// SIMATIC S7-200 SMART project (STEP 7-Micro/WIN SMART), CPU CR40

SYMBOL_TABLE 表格 1
启动               M0.4
延时启动             M0.5
延时装置             T37
工件夹持检测虚拟         M0.6
END_SYMBOL_TABLE

SYMBOL_TABLE 系统符号
First_Scan_On    SM0.1    // 仅在第一个扫描周期时接通
Clock_1s         SM0.5    // 针对 1 s 的周期时间，时钟脉冲接通 0.5 s，断开 0.5 s.
END_SYMBOL_TABLE

ORGANIZATION_BLOCK MAIN:OB1
TITLE=主程序
BEGIN
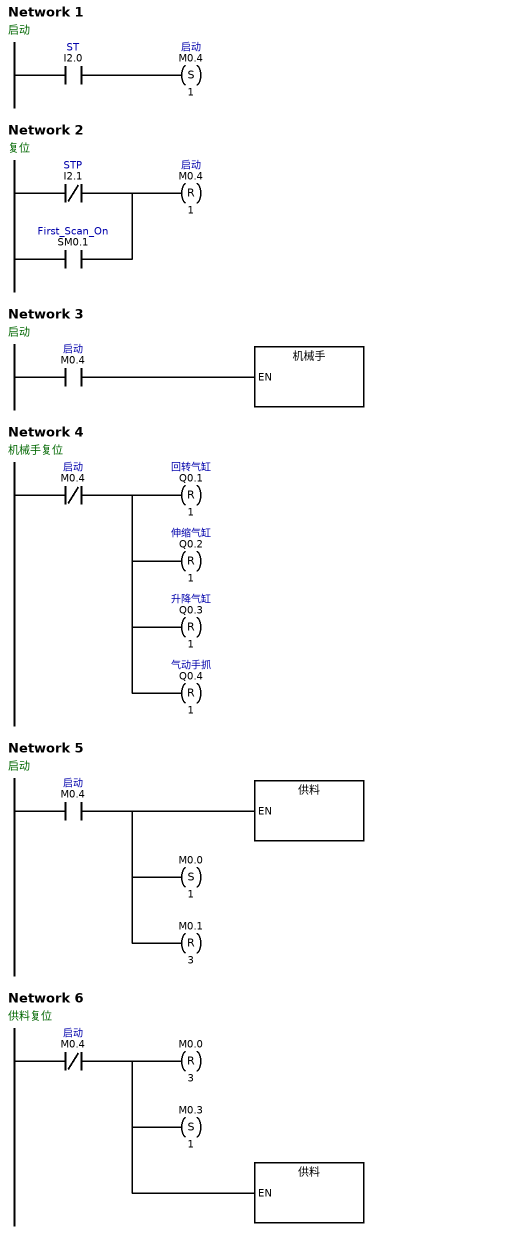
Network 1
// 启动
LD     ST:I2.0
S      启动:M0.4, 1
Network 2
// 复位
LDN    STP:I2.1
O      First_Scan_On:SM0.1
R      启动:M0.4, 1
Network 3
// 启动
LD     启动:M0.4
CALL   机械手:SBR0
Network 4
// 机械手复位
LDN    启动:M0.4
R      回转气缸:Q0.1, 1
R      伸缩气缸:Q0.2, 1
R      升降气缸:Q0.3, 1
R      气动手抓:Q0.4, 1
Network 5
// 启动
LD     启动:M0.4
CALL   供料:SBR3
S      M0.0, 1
R      M0.1, 3
Network 6
// 供料复位
LDN    启动:M0.4
R      M0.0, 3
S      M0.3, 1
CALL   供料:SBR3
END_ORGANIZATION_BLOCK

SUBROUTINE_BLOCK 机械手:SBR0
TITLE=子程序注释
BEGIN
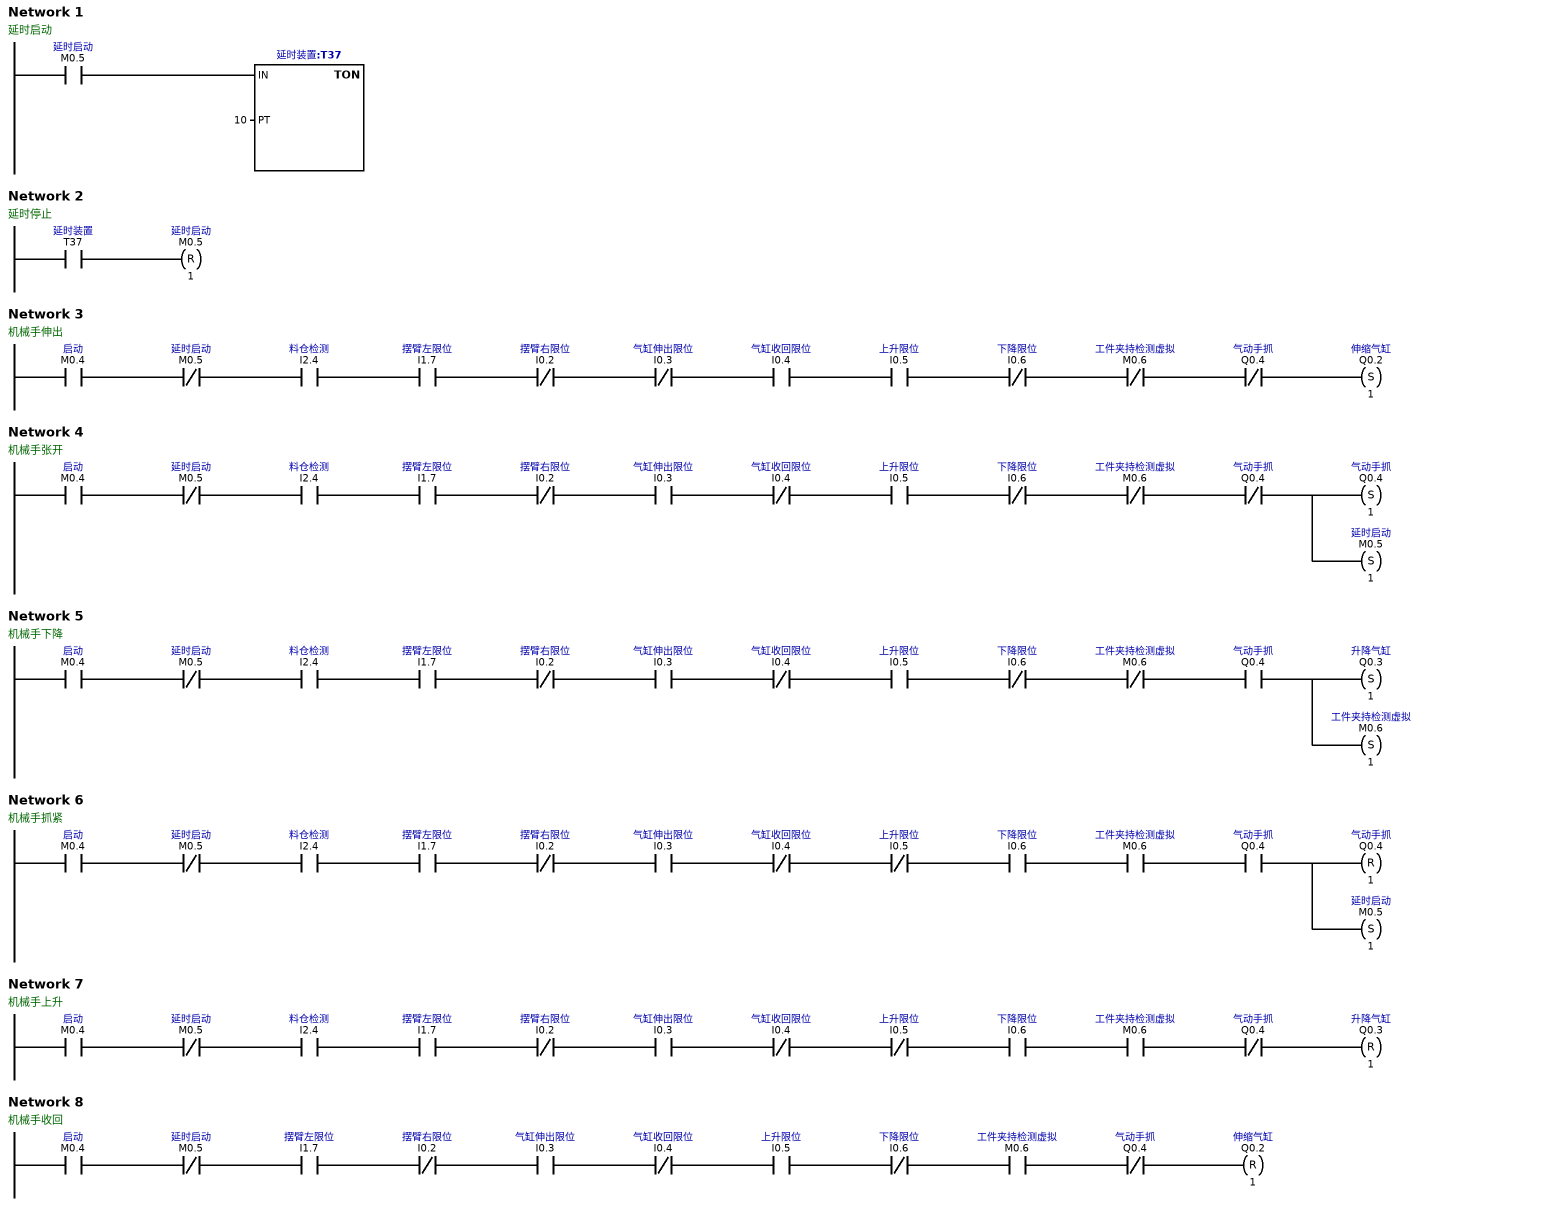
Network 1
// 延时启动
LD     延时启动:M0.5
TON    延时装置:T37, 10
Network 2
// 延时停止
LD     延时装置:T37
R      延时启动:M0.5, 1
Network 3
// 机械手伸出
LD     启动:M0.4
AN     延时启动:M0.5
A      料仓检测:I2.4
A      摆臂左限位:I1.7
AN     摆臂右限位:I0.2
AN     气缸伸出限位:I0.3
A      气缸收回限位:I0.4
A      上升限位:I0.5
AN     下降限位:I0.6
AN     工件夹持检测虚拟:M0.6
AN     气动手抓:Q0.4
S      伸缩气缸:Q0.2, 1
Network 4
// 机械手张开
LD     启动:M0.4
AN     延时启动:M0.5
A      料仓检测:I2.4
A      摆臂左限位:I1.7
AN     摆臂右限位:I0.2
A      气缸伸出限位:I0.3
AN     气缸收回限位:I0.4
A      上升限位:I0.5
AN     下降限位:I0.6
AN     工件夹持检测虚拟:M0.6
AN     气动手抓:Q0.4
S      气动手抓:Q0.4, 1
S      延时启动:M0.5, 1
Network 5
// 机械手下降
LD     启动:M0.4
AN     延时启动:M0.5
A      料仓检测:I2.4
A      摆臂左限位:I1.7
AN     摆臂右限位:I0.2
A      气缸伸出限位:I0.3
AN     气缸收回限位:I0.4
A      上升限位:I0.5
AN     下降限位:I0.6
AN     工件夹持检测虚拟:M0.6
A      气动手抓:Q0.4
S      升降气缸:Q0.3, 1
S      工件夹持检测虚拟:M0.6, 1
Network 6
// 机械手抓紧
LD     启动:M0.4
AN     延时启动:M0.5
A      料仓检测:I2.4
A      摆臂左限位:I1.7
AN     摆臂右限位:I0.2
A      气缸伸出限位:I0.3
AN     气缸收回限位:I0.4
AN     上升限位:I0.5
A      下降限位:I0.6
A      工件夹持检测虚拟:M0.6
A      气动手抓:Q0.4
R      气动手抓:Q0.4, 1
S      延时启动:M0.5, 1
Network 7
// 机械手上升
LD     启动:M0.4
AN     延时启动:M0.5
A      料仓检测:I2.4
A      摆臂左限位:I1.7
AN     摆臂右限位:I0.2
A      气缸伸出限位:I0.3
AN     气缸收回限位:I0.4
AN     上升限位:I0.5
A      下降限位:I0.6
A      工件夹持检测虚拟:M0.6
AN     气动手抓:Q0.4
R      升降气缸:Q0.3, 1
Network 8
// 机械手收回
LD     启动:M0.4
AN     延时启动:M0.5
A      摆臂左限位:I1.7
AN     摆臂右限位:I0.2
A      气缸伸出限位:I0.3
AN     气缸收回限位:I0.4
A      上升限位:I0.5
AN     下降限位:I0.6
A      工件夹持检测虚拟:M0.6
AN     气动手抓:Q0.4
R      伸缩气缸:Q0.2, 1
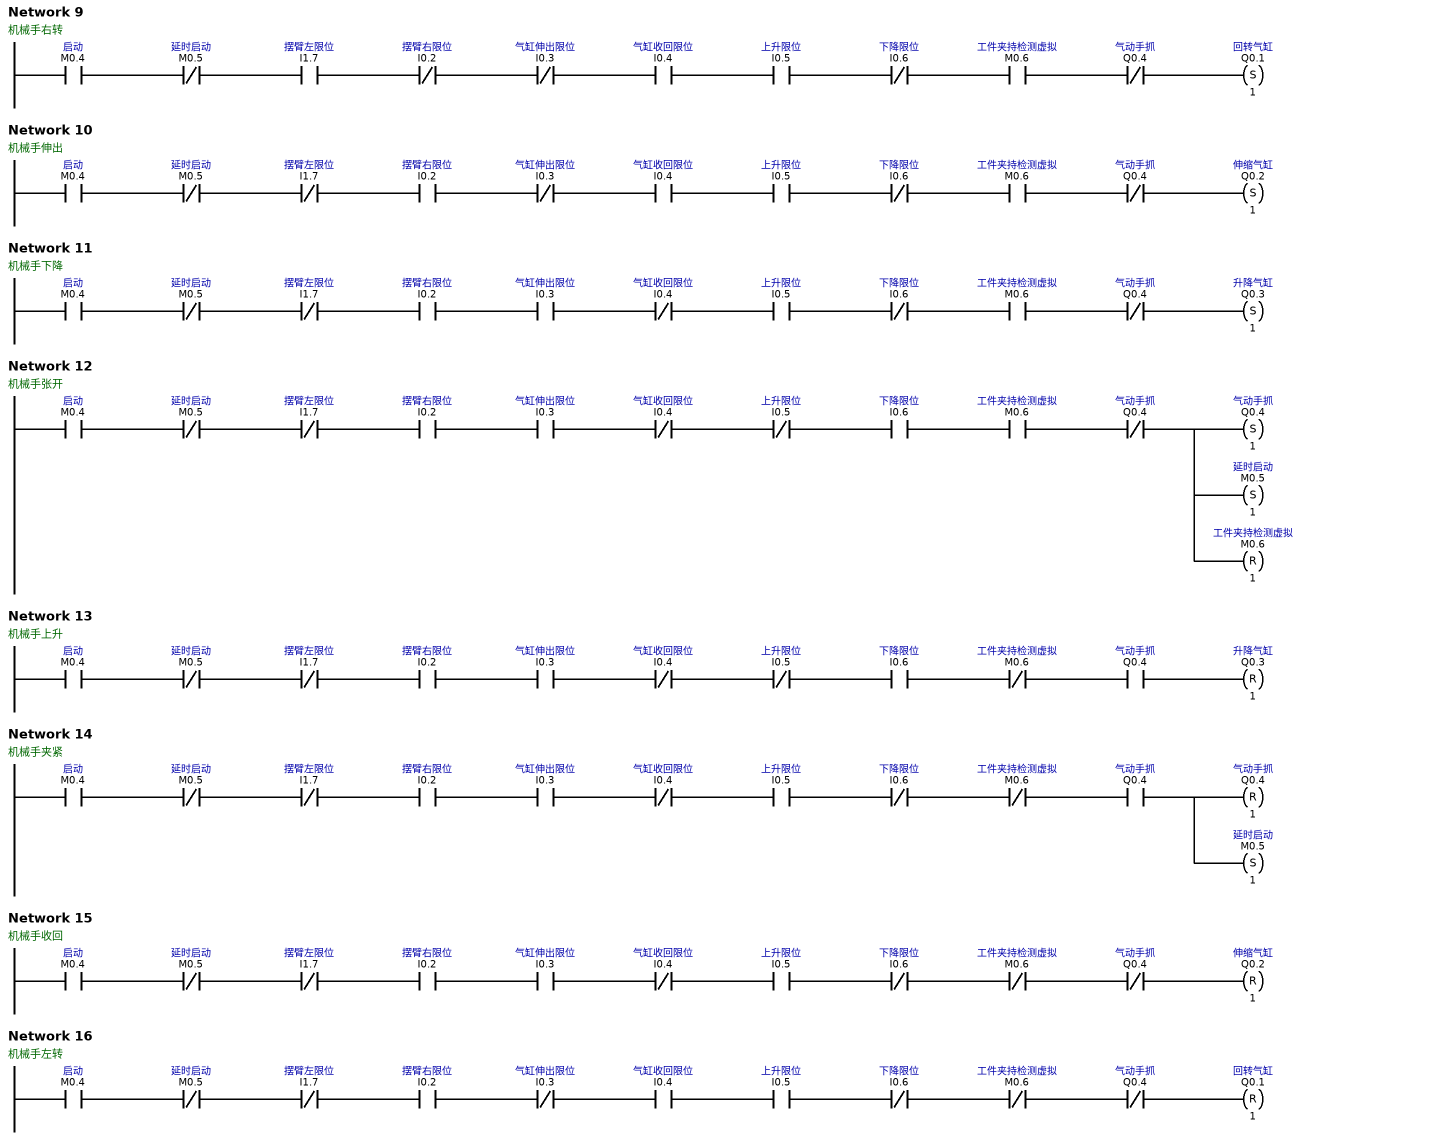
Network 9
// 机械手右转
LD     启动:M0.4
AN     延时启动:M0.5
A      摆臂左限位:I1.7
AN     摆臂右限位:I0.2
AN     气缸伸出限位:I0.3
A      气缸收回限位:I0.4
A      上升限位:I0.5
AN     下降限位:I0.6
A      工件夹持检测虚拟:M0.6
AN     气动手抓:Q0.4
S      回转气缸:Q0.1, 1
Network 10
// 机械手伸出
LD     启动:M0.4
AN     延时启动:M0.5
AN     摆臂左限位:I1.7
A      摆臂右限位:I0.2
AN     气缸伸出限位:I0.3
A      气缸收回限位:I0.4
A      上升限位:I0.5
AN     下降限位:I0.6
A      工件夹持检测虚拟:M0.6
AN     气动手抓:Q0.4
S      伸缩气缸:Q0.2, 1
Network 11
// 机械手下降
LD     启动:M0.4
AN     延时启动:M0.5
AN     摆臂左限位:I1.7
A      摆臂右限位:I0.2
A      气缸伸出限位:I0.3
AN     气缸收回限位:I0.4
A      上升限位:I0.5
AN     下降限位:I0.6
A      工件夹持检测虚拟:M0.6
AN     气动手抓:Q0.4
S      升降气缸:Q0.3, 1
Network 12
// 机械手张开
LD     启动:M0.4
AN     延时启动:M0.5
AN     摆臂左限位:I1.7
A      摆臂右限位:I0.2
A      气缸伸出限位:I0.3
AN     气缸收回限位:I0.4
AN     上升限位:I0.5
A      下降限位:I0.6
A      工件夹持检测虚拟:M0.6
AN     气动手抓:Q0.4
S      气动手抓:Q0.4, 1
S      延时启动:M0.5, 1
R      工件夹持检测虚拟:M0.6, 1
Network 13
// 机械手上升
LD     启动:M0.4
AN     延时启动:M0.5
AN     摆臂左限位:I1.7
A      摆臂右限位:I0.2
A      气缸伸出限位:I0.3
AN     气缸收回限位:I0.4
AN     上升限位:I0.5
A      下降限位:I0.6
AN     工件夹持检测虚拟:M0.6
A      气动手抓:Q0.4
R      升降气缸:Q0.3, 1
Network 14
// 机械手夹紧
LD     启动:M0.4
AN     延时启动:M0.5
AN     摆臂左限位:I1.7
A      摆臂右限位:I0.2
A      气缸伸出限位:I0.3
AN     气缸收回限位:I0.4
A      上升限位:I0.5
AN     下降限位:I0.6
AN     工件夹持检测虚拟:M0.6
A      气动手抓:Q0.4
R      气动手抓:Q0.4, 1
S      延时启动:M0.5, 1
Network 15
// 机械手收回
LD     启动:M0.4
AN     延时启动:M0.5
AN     摆臂左限位:I1.7
A      摆臂右限位:I0.2
A      气缸伸出限位:I0.3
AN     气缸收回限位:I0.4
A      上升限位:I0.5
AN     下降限位:I0.6
AN     工件夹持检测虚拟:M0.6
AN     气动手抓:Q0.4
R      伸缩气缸:Q0.2, 1
Network 16
// 机械手左转
LD     启动:M0.4
AN     延时启动:M0.5
AN     摆臂左限位:I1.7
A      摆臂右限位:I0.2
AN     气缸伸出限位:I0.3
A      气缸收回限位:I0.4
A      上升限位:I0.5
AN     下降限位:I0.6
AN     工件夹持检测虚拟:M0.6
AN     气动手抓:Q0.4
R      回转气缸:Q0.1, 1
END_SUBROUTINE_BLOCK

SUBROUTINE_BLOCK 供料:SBR3
TITLE=M0.0 绿灯常亮，电机运行
// M0.1 绿灯闪烁，电机停止
// M0.2 黄灯闪烁，电机停止
// M0.3 红灯常亮，电机停止
BEGIN
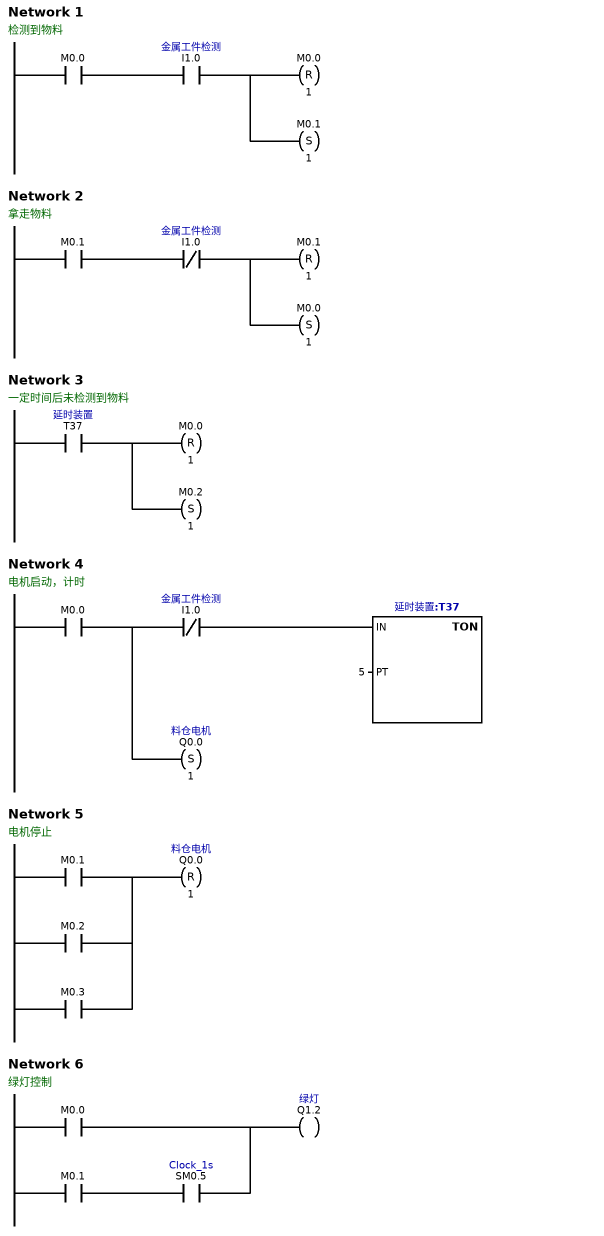
Network 1
// 检测到物料
LD     M0.0
A      金属工件检测:I1.0
R      M0.0, 1
S      M0.1, 1
Network 2
// 拿走物料
LD     M0.1
AN     金属工件检测:I1.0
R      M0.1, 1
S      M0.0, 1
Network 3
// 一定时间后未检测到物料
LD     延时装置:T37
R      M0.0, 1
S      M0.2, 1
Network 4
// 电机启动，计时
LD     M0.0
LPS
AN     金属工件检测:I1.0
TON    延时装置:T37, 5
LPP
S      料仓电机:Q0.0, 1
Network 5
// 电机停止
LD     M0.1
O      M0.2
O      M0.3
R      料仓电机:Q0.0, 1
Network 6
// 绿灯控制
LD     M0.0
LD     M0.1
A      Clock_1s:SM0.5
OLD
=      绿灯:Q1.2
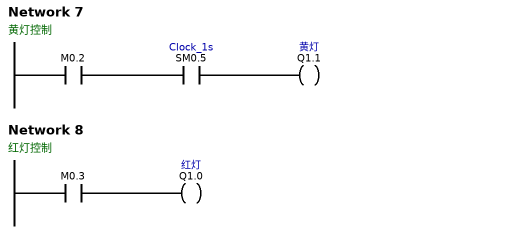
Network 7
// 黄灯控制
LD     M0.2
A      Clock_1s:SM0.5
=      黄灯:Q1.1
Network 8
// 红灯控制
LD     M0.3
=      红灯:Q1.0
END_SUBROUTINE_BLOCK
